// TIA Portal project "WpfPlcMonitor" (V17)

(* hardware
DEVICE "S7-1200 station_1"  S7-1200 Station
   slot 0: "Rack_0"  S7-1200 Rack  Rack  V1.0
   slot 1: "PLC_1"  CPU 1214C DC/DC/DC  6ES7 214-1AG40-0XB0  V4.5
*)

// ===== PLC "PLC_1"  CPU 1214C DC/DC/DC =====

DATA_BLOCK "数据块_1"   // DB1
{ S7_Optimized_Access := 'FALSE' }
VERSION : 0.1
   VAR
      Temperature : Real := 25.0;   // 实时温度
      Humidity : Real := 50.0;   // 实时湿度
      RunStatus : Bool := true;   // 设备运行状态
      Angle : Real := 0.0;   // 内部正弦计算角度
   END_VAR
BEGIN
END_DATA_BLOCK

ORGANIZATION_BLOCK "Main"   // OB1, LAD, ProgramCycle
TITLE = "Main Program Sweep (Cycle)"
{ S7_Optimized_Access := 'TRUE' }
VERSION : 0.1
   VAR_INPUT
      Initial_Call : Bool;   // Initial call of this OB
      Remanence : Bool;   // =True, if remanent data are available
   END_VAR
BEGIN

REGION Network 1 (SCL): 模拟数据
   // 1. 累加角度（用于生成平滑的工艺正弦波）
   "数据块_1".Angle := "数据块_1".Angle + 0.02;
   IF "数据块_1".Angle >= 6.283185 THEN
       "数据块_1".Angle := 0.0;
   END_IF;

   // 2. 利用 SIN/COS 函数计算温湿度（模拟正常的工艺波动范围）
   "数据块_1".Temperature := 25.0 + 5.0 * SIN(IN := "数据块_1".Angle);
   "数据块_1".Humidity := 60.0 + 20.0 * COS(IN := "数据块_1".Angle);

   // 3. 基础运行状态默认给常态 TRUE（运行中）
   "数据块_1".RunStatus := TRUE;

   // 4. 工业级超温保护逻辑：当温度超过 31.5℃ 时，触发安全停机
   IF "数据块_1".Temperature > 31.5 THEN
       "数据块_1".RunStatus := FALSE; // 超温时置为 FALSE（停止/报警保护）
   END_IF;
END_REGION
END_ORGANIZATION_BLOCK